// Mitsubishi GX Works2 project: GX W2 L6 Ex 1 DK C   PLC: FX3G

// global labels: Global1
VAR_GLOBAL
  iStart_PB AT X001 : BOOL;
  oO_Letter AT Y001 : BOOL;
  oP_Letter AT Y002 : BOOL;
  oE_Letter AT Y003 : BOOL;
  oN_Letter AT Y004 : BOOL;
  iOn_Switch AT X002 : BOOL;
  oBorder AT Y000 : BOOL;
END_VAR

// task Task_01 (event TRUE, interval 0, priority 31): POU_01

PROGRAM POU_01
VAR
  wSequence_States : INT;
  TON_1 : TON;
  TON_2 : TON;
  TON_3 : TON;
  TON_4 : TON;
END_VAR
(* structured ladder/FBD written out as ST: instructions are called as NAME(EN, inputs, outputs); _pN, _eN, _tN stand for wires *)
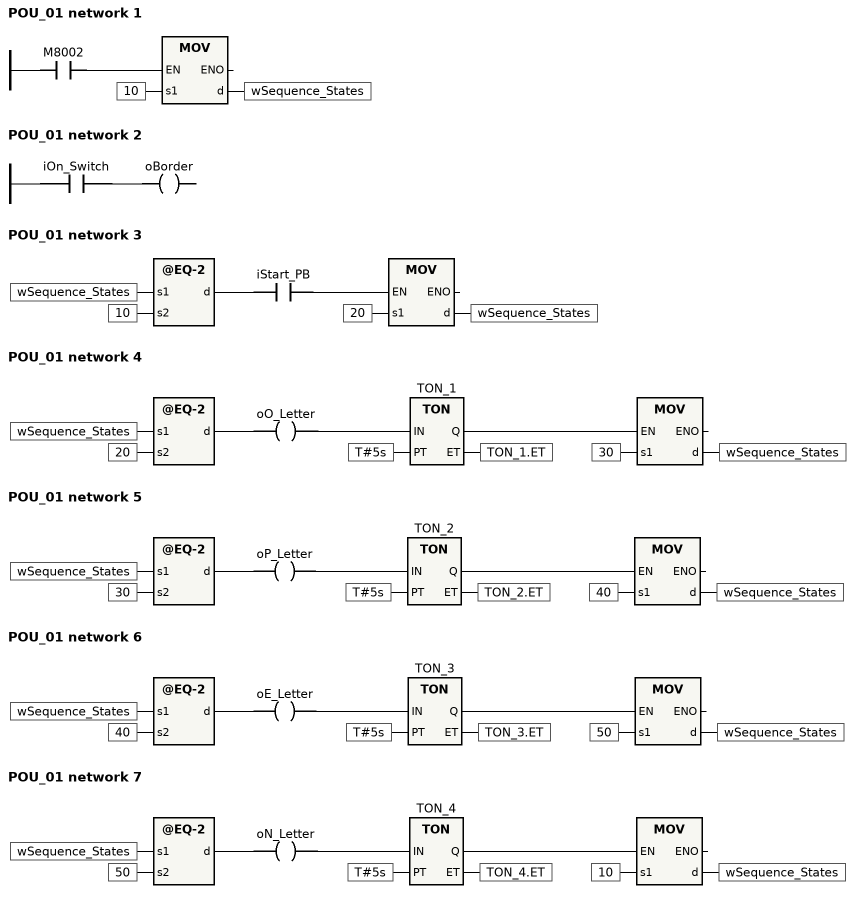
(* network 1 *)
MOV(M8002, 10, wSequence_States);
(* network 2 *)
oBorder := iOn_Switch;
(* network 3 *)
MOV(@EQ-2(wSequence_States, 10) AND iStart_PB, 20, wSequence_States);
(* network 4 *)
_p1 := @EQ-2(wSequence_States, 20);
oO_Letter := _p1;
TON_1(IN := _p1, PT := T#5s, ET => TON_1.ET);
MOV(TON_1.Q, 30, wSequence_States);
(* network 5 *)
_p1 := @EQ-2(wSequence_States, 30);
oP_Letter := _p1;
TON_2(IN := _p1, PT := T#5s, ET => TON_2.ET);
MOV(TON_2.Q, 40, wSequence_States);
(* network 6 *)
_p1 := @EQ-2(wSequence_States, 40);
oE_Letter := _p1;
TON_3(IN := _p1, PT := T#5s, ET => TON_3.ET);
MOV(TON_3.Q, 50, wSequence_States);
(* network 7 *)
_p1 := @EQ-2(wSequence_States, 50);
oN_Letter := _p1;
TON_4(IN := _p1, PT := T#5s, ET => TON_4.ET);
MOV(TON_4.Q, 10, wSequence_States);
END_PROGRAM
